FUNCTION "RS485_2" : VOID	// FC 2
VERSION : 0.1
BEGIN
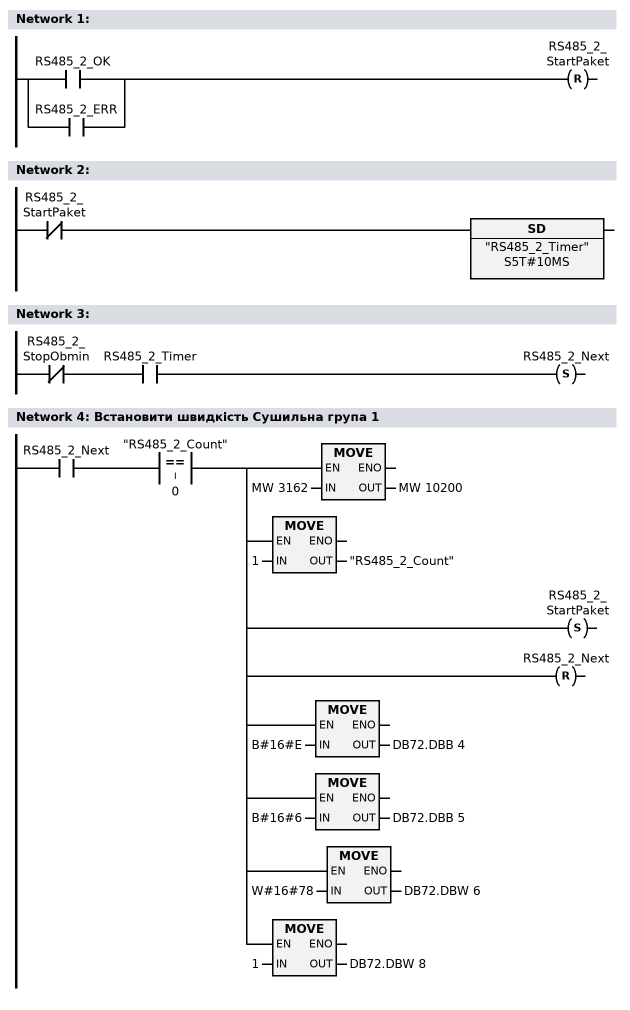
NETWORK
TITLE =
      O     "RS485_2_OK";
      O     "RS485_2_ERR";
      R     "RS485_2_StartPaket";
NETWORK
TITLE =
      AN    "RS485_2_StartPaket";
      L     S5T#10MS;
      SD    "RS485_2_Timer";
NETWORK
TITLE =
      AN    "RS485_2_StopObmin";
      A     "RS485_2_Timer";
      S     "RS485_2_Next";
NETWORK
TITLE = Встановити швидкість Сушильна група 1
      A     "RS485_2_Next";
      A(;
      L     "RS485_2_Count";
      L     0;
      ==I;
      );
      =     L 0.0;
      A     L 0.0;
      JNB   _001;
      L     MW 3162;
      T     MW 10200;
_001: NOP   0;
      A     L 0.0;
      JNB   _002;
      L     1;
      T     "RS485_2_Count";
_002: NOP   0;
      A     L 0.0;
      BLD   102;
      S     "RS485_2_StartPaket";
      A     L 0.0;
      BLD   102;
      R     "RS485_2_Next";
      A     L 0.0;
      JNB   _003;
      L     B#16#E;
      T     DB72.DBB 4;
_003: NOP   0;
      A     L 0.0;
      JNB   _004;
      L     B#16#6;
      T     DB72.DBB 5;
_004: NOP   0;
      A     L 0.0;
      JNB   _005;
      L     W#16#78;
      T     DB72.DBW 6;
_005: NOP   0;
      A     L 0.0;
      JNB   _006;
      L     1;
      T     DB72.DBW 8;
_006: NOP   0;
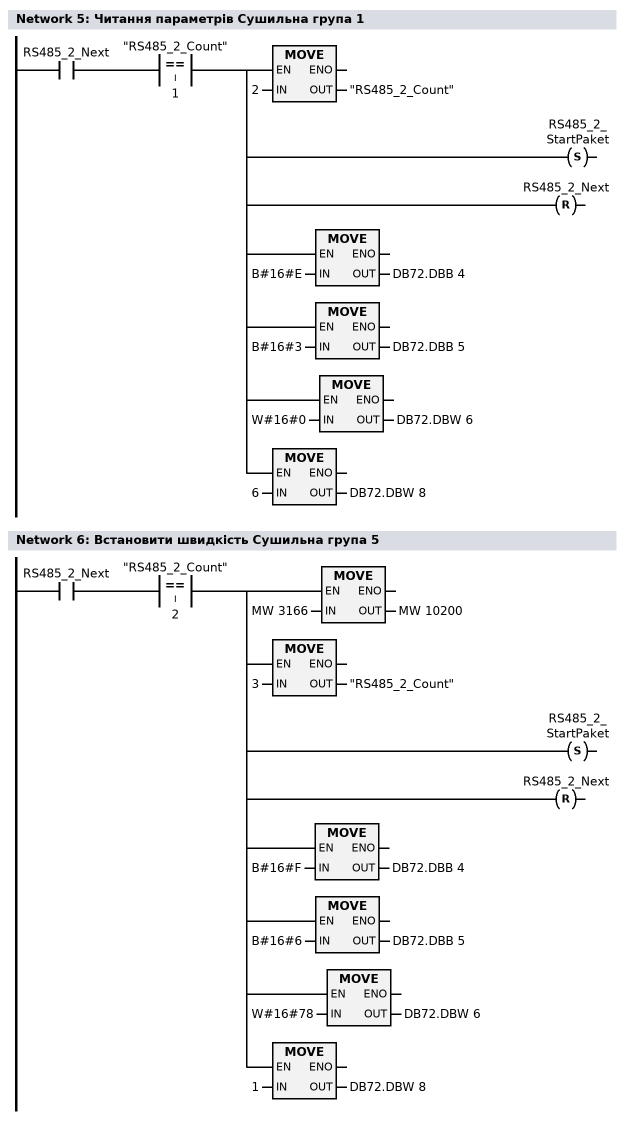
NETWORK
TITLE = Читання параметрів Сушильна група 1
      A     "RS485_2_Next";
      A(;
      L     "RS485_2_Count";
      L     1;
      ==I;
      );
      =     L 0.0;
      A     L 0.0;
      JNB   _007;
      L     2;
      T     "RS485_2_Count";
_007: NOP   0;
      A     L 0.0;
      BLD   102;
      S     "RS485_2_StartPaket";
      A     L 0.0;
      BLD   102;
      R     "RS485_2_Next";
      A     L 0.0;
      JNB   _008;
      L     B#16#E;
      T     DB72.DBB 4;
_008: NOP   0;
      A     L 0.0;
      JNB   _009;
      L     B#16#3;
      T     DB72.DBB 5;
_009: NOP   0;
      A     L 0.0;
      JNB   _00a;
      L     W#16#0;
      T     DB72.DBW 6;
_00a: NOP   0;
      A     L 0.0;
      JNB   _00b;
      L     6;
      T     DB72.DBW 8;
_00b: NOP   0;
NETWORK
TITLE = Встановити швидкість Сушильна група 5
      A     "RS485_2_Next";
      A(;
      L     "RS485_2_Count";
      L     2;
      ==I;
      );
      =     L 0.0;
      A     L 0.0;
      JNB   _00c;
      L     MW 3166;
      T     MW 10200;
_00c: NOP   0;
      A     L 0.0;
      JNB   _00d;
      L     3;
      T     "RS485_2_Count";
_00d: NOP   0;
      A     L 0.0;
      BLD   102;
      S     "RS485_2_StartPaket";
      A     L 0.0;
      BLD   102;
      R     "RS485_2_Next";
      A     L 0.0;
      JNB   _00e;
      L     B#16#F;
      T     DB72.DBB 4;
_00e: NOP   0;
      A     L 0.0;
      JNB   _00f;
      L     B#16#6;
      T     DB72.DBB 5;
_00f: NOP   0;
      A     L 0.0;
      JNB   _010;
      L     W#16#78;
      T     DB72.DBW 6;
_010: NOP   0;
      A     L 0.0;
      JNB   _011;
      L     1;
      T     DB72.DBW 8;
_011: NOP   0;
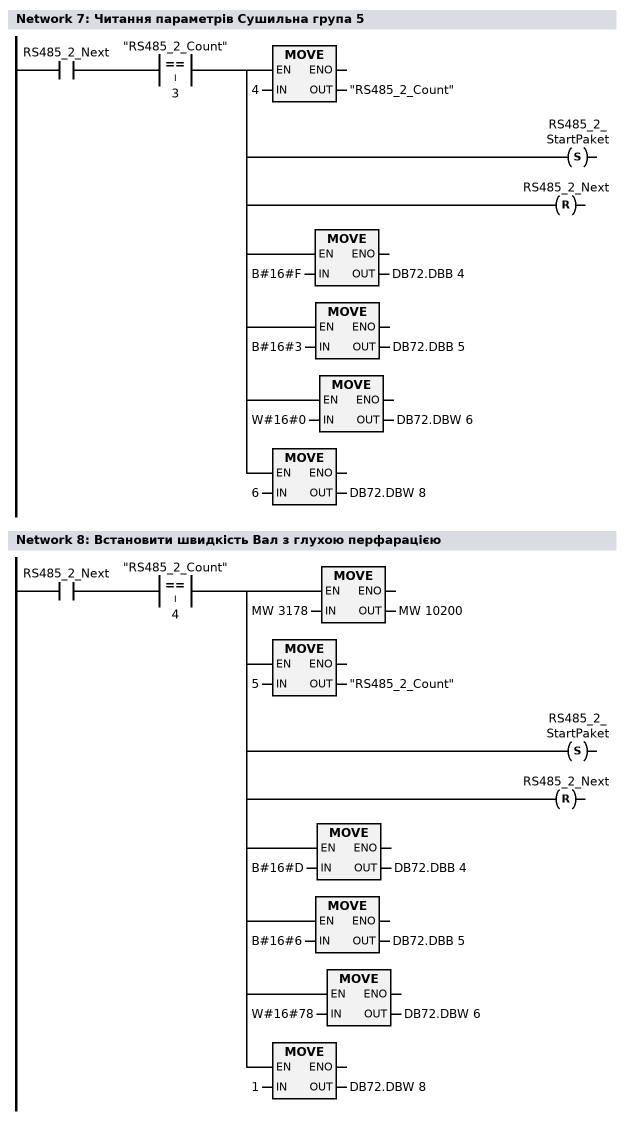
NETWORK
TITLE = Читання параметрів Сушильна група 5
      A     "RS485_2_Next";
      A(;
      L     "RS485_2_Count";
      L     3;
      ==I;
      );
      =     L 0.0;
      A     L 0.0;
      JNB   _012;
      L     4;
      T     "RS485_2_Count";
_012: NOP   0;
      A     L 0.0;
      BLD   102;
      S     "RS485_2_StartPaket";
      A     L 0.0;
      BLD   102;
      R     "RS485_2_Next";
      A     L 0.0;
      JNB   _013;
      L     B#16#F;
      T     DB72.DBB 4;
_013: NOP   0;
      A     L 0.0;
      JNB   _014;
      L     B#16#3;
      T     DB72.DBB 5;
_014: NOP   0;
      A     L 0.0;
      JNB   _015;
      L     W#16#0;
      T     DB72.DBW 6;
_015: NOP   0;
      A     L 0.0;
      JNB   _016;
      L     6;
      T     DB72.DBW 8;
_016: NOP   0;
NETWORK
TITLE = Встановити швидкість Вал з глухою перфарацією
      A     "RS485_2_Next";
      A(;
      L     "RS485_2_Count";
      L     4;
      ==I;
      );
      =     L 0.0;
      A     L 0.0;
      JNB   _017;
      L     MW 3178;
      T     MW 10200;
_017: NOP   0;
      A     L 0.0;
      JNB   _018;
      L     5;
      T     "RS485_2_Count";
_018: NOP   0;
      A     L 0.0;
      BLD   102;
      S     "RS485_2_StartPaket";
      A     L 0.0;
      BLD   102;
      R     "RS485_2_Next";
      A     L 0.0;
      JNB   _019;
      L     B#16#D;
      T     DB72.DBB 4;
_019: NOP   0;
      A     L 0.0;
      JNB   _01a;
      L     B#16#6;
      T     DB72.DBB 5;
_01a: NOP   0;
      A     L 0.0;
      JNB   _01b;
      L     W#16#78;
      T     DB72.DBW 6;
_01b: NOP   0;
      A     L 0.0;
      JNB   _01c;
      L     1;
      T     DB72.DBW 8;
_01c: NOP   0;
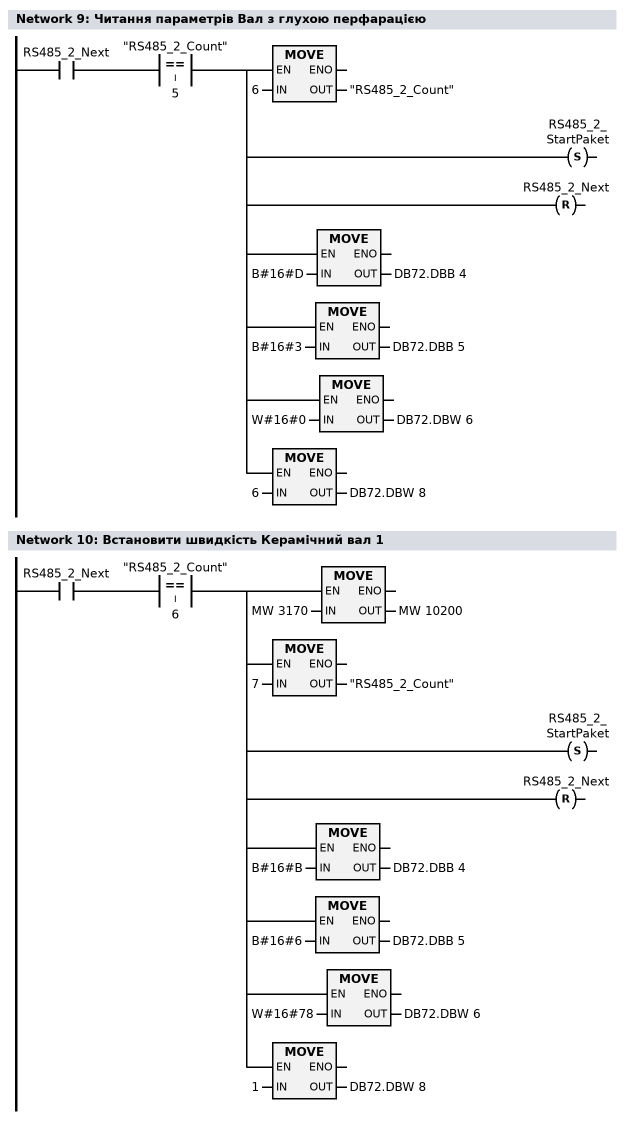
NETWORK
TITLE = Читання параметрів Вал з глухою перфарацією
      A     "RS485_2_Next";
      A(;
      L     "RS485_2_Count";
      L     5;
      ==I;
      );
      =     L 0.0;
      A     L 0.0;
      JNB   _01d;
      L     6;
      T     "RS485_2_Count";
_01d: NOP   0;
      A     L 0.0;
      BLD   102;
      S     "RS485_2_StartPaket";
      A     L 0.0;
      BLD   102;
      R     "RS485_2_Next";
      A     L 0.0;
      JNB   _01e;
      L     B#16#D;
      T     DB72.DBB 4;
_01e: NOP   0;
      A     L 0.0;
      JNB   _01f;
      L     B#16#3;
      T     DB72.DBB 5;
_01f: NOP   0;
      A     L 0.0;
      JNB   _020;
      L     W#16#0;
      T     DB72.DBW 6;
_020: NOP   0;
      A     L 0.0;
      JNB   _021;
      L     6;
      T     DB72.DBW 8;
_021: NOP   0;
NETWORK
TITLE = Встановити швидкість Керамічний вал 1
      A     "RS485_2_Next";
      A(;
      L     "RS485_2_Count";
      L     6;
      ==I;
      );
      =     L 0.0;
      A     L 0.0;
      JNB   _022;
      L     MW 3170;
      T     MW 10200;
_022: NOP   0;
      A     L 0.0;
      JNB   _023;
      L     7;
      T     "RS485_2_Count";
_023: NOP   0;
      A     L 0.0;
      BLD   102;
      S     "RS485_2_StartPaket";
      A     L 0.0;
      BLD   102;
      R     "RS485_2_Next";
      A     L 0.0;
      JNB   _024;
      L     B#16#B;
      T     DB72.DBB 4;
_024: NOP   0;
      A     L 0.0;
      JNB   _025;
      L     B#16#6;
      T     DB72.DBB 5;
_025: NOP   0;
      A     L 0.0;
      JNB   _026;
      L     W#16#78;
      T     DB72.DBW 6;
_026: NOP   0;
      A     L 0.0;
      JNB   _027;
      L     1;
      T     DB72.DBW 8;
_027: NOP   0;
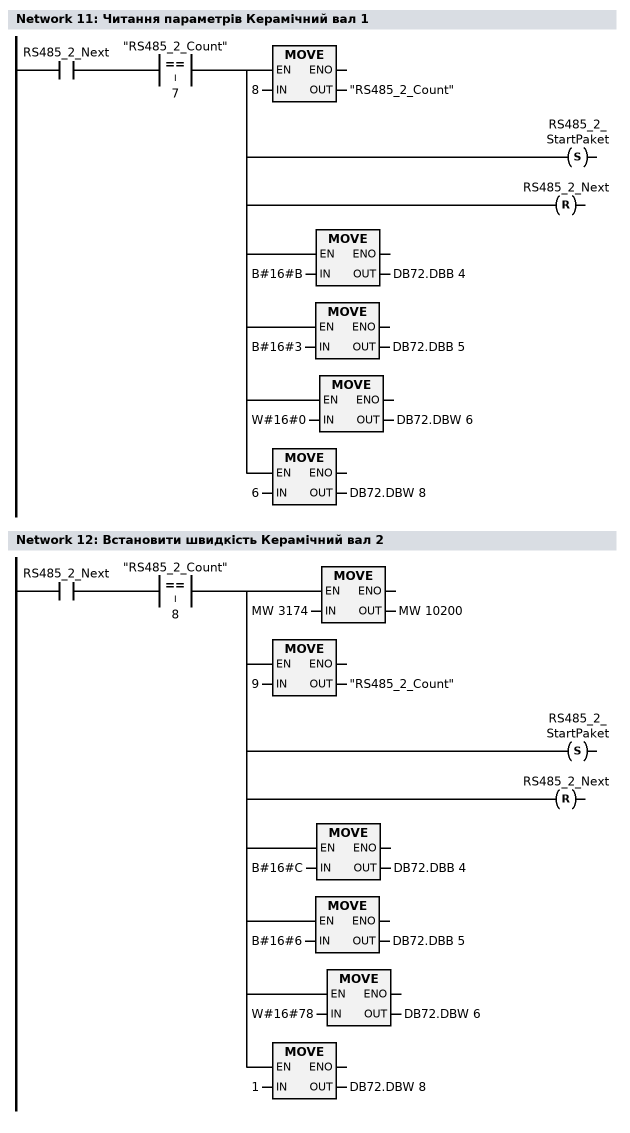
NETWORK
TITLE = Читання параметрів Керамічний вал 1
      A     "RS485_2_Next";
      A(;
      L     "RS485_2_Count";
      L     7;
      ==I;
      );
      =     L 0.0;
      A     L 0.0;
      JNB   _028;
      L     8;
      T     "RS485_2_Count";
_028: NOP   0;
      A     L 0.0;
      BLD   102;
      S     "RS485_2_StartPaket";
      A     L 0.0;
      BLD   102;
      R     "RS485_2_Next";
      A     L 0.0;
      JNB   _029;
      L     B#16#B;
      T     DB72.DBB 4;
_029: NOP   0;
      A     L 0.0;
      JNB   _02a;
      L     B#16#3;
      T     DB72.DBB 5;
_02a: NOP   0;
      A     L 0.0;
      JNB   _02b;
      L     W#16#0;
      T     DB72.DBW 6;
_02b: NOP   0;
      A     L 0.0;
      JNB   _02c;
      L     6;
      T     DB72.DBW 8;
_02c: NOP   0;
NETWORK
TITLE = Встановити швидкість Керамічний вал 2
      A     "RS485_2_Next";
      A(;
      L     "RS485_2_Count";
      L     8;
      ==I;
      );
      =     L 0.0;
      A     L 0.0;
      JNB   _046;
      L     MW 3174;
      T     MW 10200;
_046: NOP   0;
      A     L 0.0;
      JNB   _047;
      L     9;
      T     "RS485_2_Count";
_047: NOP   0;
      A     L 0.0;
      BLD   102;
      S     "RS485_2_StartPaket";
      A     L 0.0;
      BLD   102;
      R     "RS485_2_Next";
      A     L 0.0;
      JNB   _048;
      L     B#16#C;
      T     DB72.DBB 4;
_048: NOP   0;
      A     L 0.0;
      JNB   _049;
      L     B#16#6;
      T     DB72.DBB 5;
_049: NOP   0;
      A     L 0.0;
      JNB   _04a;
      L     W#16#78;
      T     DB72.DBW 6;
_04a: NOP   0;
      A     L 0.0;
      JNB   _04b;
      L     1;
      T     DB72.DBW 8;
_04b: NOP   0;
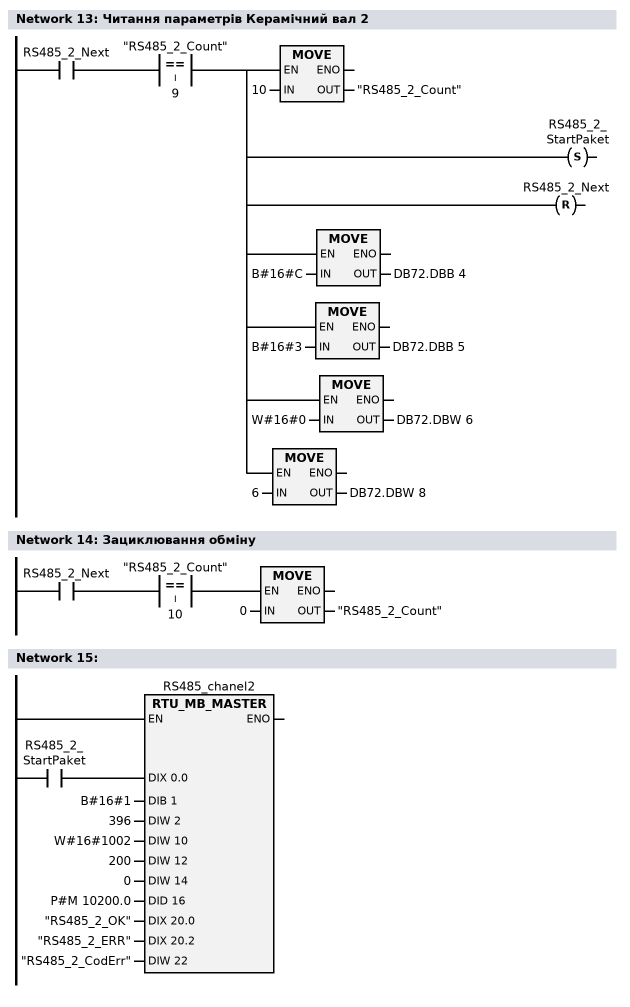
NETWORK
TITLE = Читання параметрів Керамічний вал 2
      A     "RS485_2_Next";
      A(;
      L     "RS485_2_Count";
      L     9;
      ==I;
      );
      =     L 0.0;
      A     L 0.0;
      JNB   _04c;
      L     10;
      T     "RS485_2_Count";
_04c: NOP   0;
      A     L 0.0;
      BLD   102;
      S     "RS485_2_StartPaket";
      A     L 0.0;
      BLD   102;
      R     "RS485_2_Next";
      A     L 0.0;
      JNB   _04d;
      L     B#16#C;
      T     DB72.DBB 4;
_04d: NOP   0;
      A     L 0.0;
      JNB   _04e;
      L     B#16#3;
      T     DB72.DBB 5;
_04e: NOP   0;
      A     L 0.0;
      JNB   _04f;
      L     W#16#0;
      T     DB72.DBW 6;
_04f: NOP   0;
      A     L 0.0;
      JNB   _050;
      L     6;
      T     DB72.DBW 8;
_050: NOP   0;
NETWORK
TITLE = Зациклювання обміну
      A     "RS485_2_Next";
      A(;
      L     "RS485_2_Count";
      L     10;
      ==I;
      );
      JNB   _051;
      L     0;
      T     "RS485_2_Count";
_051: NOP   0;
NETWORK
TITLE =
      A     "RS485_2_StartPaket";
      =     L 0.0;
      BLD   103;
      CALL  "RTU_MB_MASTER" , "RS485_chanel2" (
           DIX 0.0                  := L 0.0,
           DIB 1                    := B#16#1,
           DIW 2                    := 396,
           DIW 10                   := W#16#1002,
           DIW 12                   := 200,
           DIW 14                   := 0,
           DID 16                   := P#M 10200.0,
           DIX 20.0                 := "RS485_2_OK",
           DIX 20.2                 := "RS485_2_ERR",
           DIW 22                   := "RS485_2_CodErr");
      NOP   0;
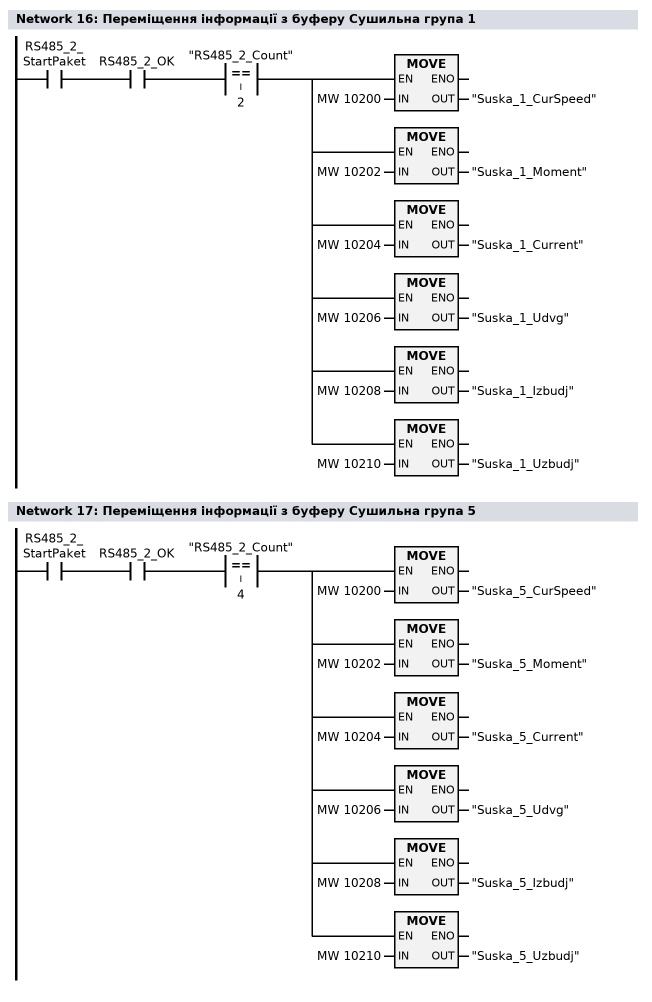
NETWORK
TITLE = Переміщення інформації з буферу Сушильна група 1
      A     "RS485_2_StartPaket";
      A     "RS485_2_OK";
      A(;
      L     "RS485_2_Count";
      L     2;
      ==I;
      );
      =     L 0.0;
      A     L 0.0;
      JNB   _052;
      L     MW 10200;
      T     "Suska_1_CurSpeed";
_052: NOP   0;
      A     L 0.0;
      JNB   _053;
      L     MW 10202;
      T     "Suska_1_Moment";
_053: NOP   0;
      A     L 0.0;
      JNB   _054;
      L     MW 10204;
      T     "Suska_1_Current";
_054: NOP   0;
      A     L 0.0;
      JNB   _055;
      L     MW 10206;
      T     "Suska_1_Udvg";
_055: NOP   0;
      A     L 0.0;
      JNB   _056;
      L     MW 10208;
      T     "Suska_1_Izbudj";
_056: NOP   0;
      A     L 0.0;
      JNB   _057;
      L     MW 10210;
      T     "Suska_1_Uzbudj";
_057: NOP   0;
NETWORK
TITLE = Переміщення інформації з буферу Сушильна група 5
      A     "RS485_2_StartPaket";
      A     "RS485_2_OK";
      A(;
      L     "RS485_2_Count";
      L     4;
      ==I;
      );
      =     L 0.0;
      A     L 0.0;
      JNB   _058;
      L     MW 10200;
      T     "Suska_5_CurSpeed";
_058: NOP   0;
      A     L 0.0;
      JNB   _059;
      L     MW 10202;
      T     "Suska_5_Moment";
_059: NOP   0;
      A     L 0.0;
      JNB   _05a;
      L     MW 10204;
      T     "Suska_5_Current";
_05a: NOP   0;
      A     L 0.0;
      JNB   _05b;
      L     MW 10206;
      T     "Suska_5_Udvg";
_05b: NOP   0;
      A     L 0.0;
      JNB   _05c;
      L     MW 10208;
      T     "Suska_5_Izbudj";
_05c: NOP   0;
      A     L 0.0;
      JNB   _05d;
      L     MW 10210;
      T     "Suska_5_Uzbudj";
_05d: NOP   0;
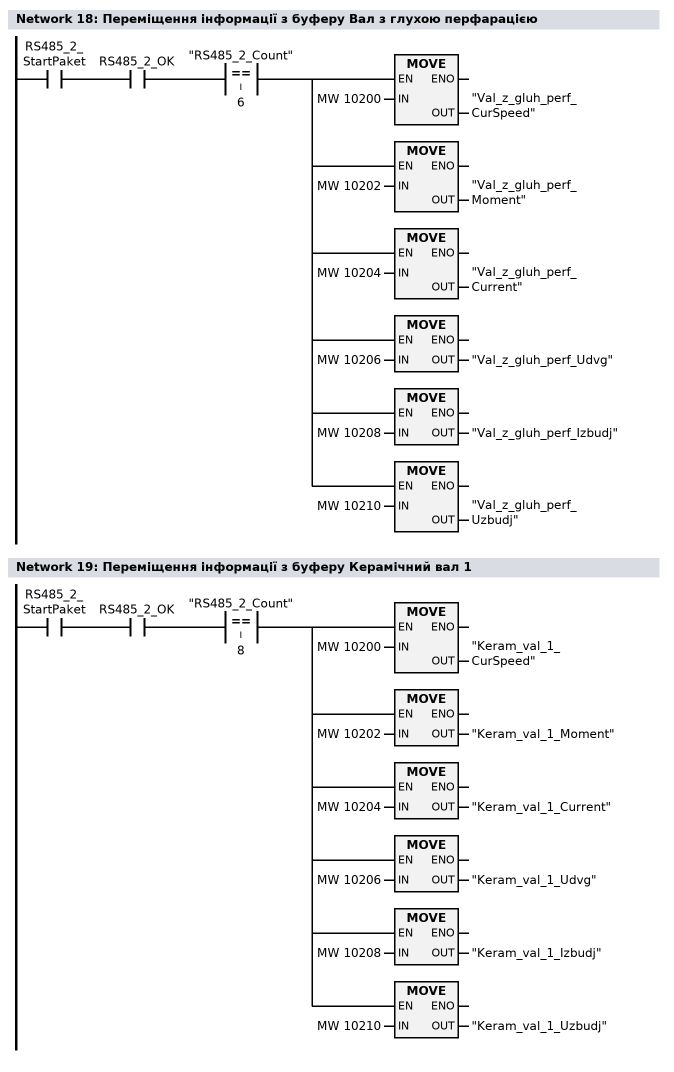
NETWORK
TITLE = Переміщення інформації з буферу Вал з глухою перфарацією
      A     "RS485_2_StartPaket";
      A     "RS485_2_OK";
      A(;
      L     "RS485_2_Count";
      L     6;
      ==I;
      );
      =     L 0.0;
      A     L 0.0;
      JNB   _05e;
      L     MW 10200;
      T     "Val_z_gluh_perf_CurSpeed";
_05e: NOP   0;
      A     L 0.0;
      JNB   _05f;
      L     MW 10202;
      T     "Val_z_gluh_perf_Moment";
_05f: NOP   0;
      A     L 0.0;
      JNB   _060;
      L     MW 10204;
      T     "Val_z_gluh_perf_Current";
_060: NOP   0;
      A     L 0.0;
      JNB   _061;
      L     MW 10206;
      T     "Val_z_gluh_perf_Udvg";
_061: NOP   0;
      A     L 0.0;
      JNB   _062;
      L     MW 10208;
      T     "Val_z_gluh_perf_Izbudj";
_062: NOP   0;
      A     L 0.0;
      JNB   _063;
      L     MW 10210;
      T     "Val_z_gluh_perf_Uzbudj";
_063: NOP   0;
NETWORK
TITLE = Переміщення інформації з буферу Керамічний вал 1
      A     "RS485_2_StartPaket";
      A     "RS485_2_OK";
      A(;
      L     "RS485_2_Count";
      L     8;
      ==I;
      );
      =     L 0.0;
      A     L 0.0;
      JNB   _064;
      L     MW 10200;
      T     "Keram_val_1_CurSpeed";
_064: NOP   0;
      A     L 0.0;
      JNB   _065;
      L     MW 10202;
      T     "Keram_val_1_Moment";
_065: NOP   0;
      A     L 0.0;
      JNB   _066;
      L     MW 10204;
      T     "Keram_val_1_Current";
_066: NOP   0;
      A     L 0.0;
      JNB   _067;
      L     MW 10206;
      T     "Keram_val_1_Udvg";
_067: NOP   0;
      A     L 0.0;
      JNB   _068;
      L     MW 10208;
      T     "Keram_val_1_Izbudj";
_068: NOP   0;
      A     L 0.0;
      JNB   _069;
      L     MW 10210;
      T     "Keram_val_1_Uzbudj";
_069: NOP   0;
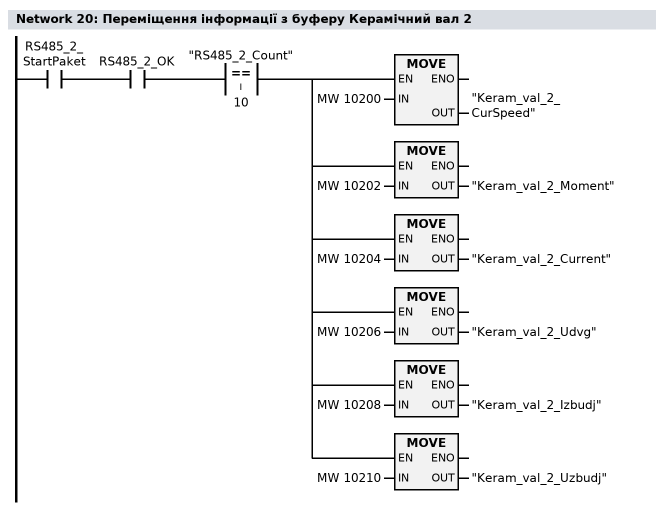
NETWORK
TITLE = Переміщення інформації з буферу Керамічний вал 2
      A     "RS485_2_StartPaket";
      A     "RS485_2_OK";
      A(;
      L     "RS485_2_Count";
      L     10;
      ==I;
      );
      =     L 0.0;
      A     L 0.0;
      JNB   _06a;
      L     MW 10200;
      T     "Keram_val_2_CurSpeed";
_06a: NOP   0;
      A     L 0.0;
      JNB   _06b;
      L     MW 10202;
      T     "Keram_val_2_Moment";
_06b: NOP   0;
      A     L 0.0;
      JNB   _06c;
      L     MW 10204;
      T     "Keram_val_2_Current";
_06c: NOP   0;
      A     L 0.0;
      JNB   _06d;
      L     MW 10206;
      T     "Keram_val_2_Udvg";
_06d: NOP   0;
      A     L 0.0;
      JNB   _06e;
      L     MW 10208;
      T     "Keram_val_2_Izbudj";
_06e: NOP   0;
      A     L 0.0;
      JNB   _06f;
      L     MW 10210;
      T     "Keram_val_2_Uzbudj";
_06f: NOP   0;
END_FUNCTION

FUNCTION "RS485_Runchanel3" : VOID	// FC 3
VERSION : 0.1
BEGIN
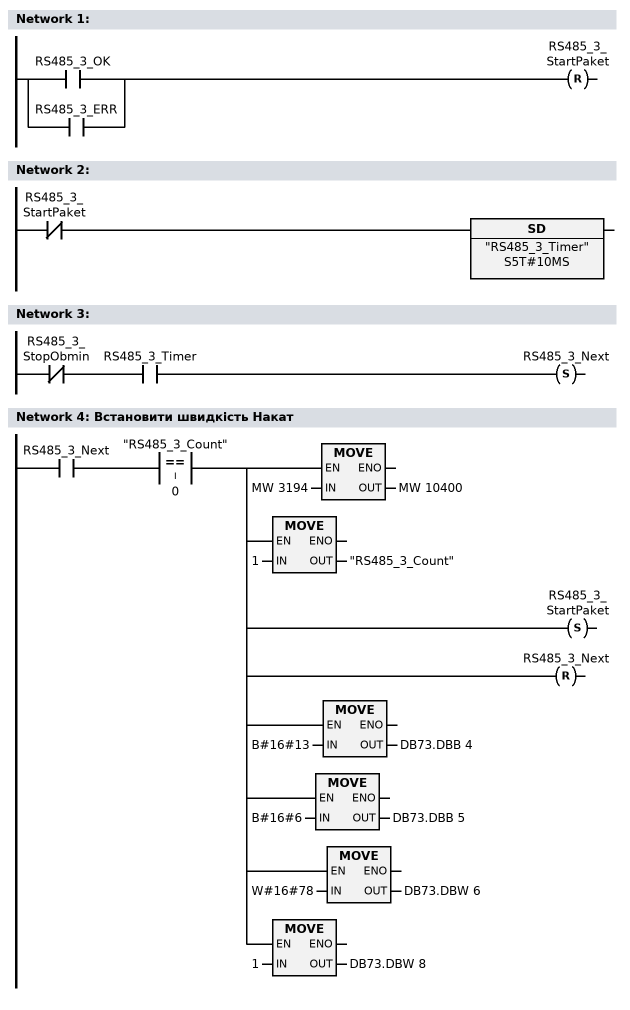
NETWORK
TITLE =
      O     "RS485_3_OK";
      O     "RS485_3_ERR";
      R     "RS485_3_StartPaket";
NETWORK
TITLE =
      AN    "RS485_3_StartPaket";
      L     S5T#10MS;
      SD    "RS485_3_Timer";
NETWORK
TITLE =
      AN    "RS485_3_StopObmin";
      A     "RS485_3_Timer";
      S     "RS485_3_Next";
NETWORK
TITLE = Встановити швидкість Накат
      A     "RS485_3_Next";
      A(;
      L     "RS485_3_Count";
      L     0;
      ==I;
      );
      =     L 0.0;
      A     L 0.0;
      JNB   _001;
      L     MW 3194;
      T     MW 10400;
_001: NOP   0;
      A     L 0.0;
      JNB   _002;
      L     1;
      T     "RS485_3_Count";
_002: NOP   0;
      A     L 0.0;
      BLD   102;
      S     "RS485_3_StartPaket";
      A     L 0.0;
      BLD   102;
      R     "RS485_3_Next";
      A     L 0.0;
      JNB   _003;
      L     B#16#13;
      T     DB73.DBB 4;
_003: NOP   0;
      A     L 0.0;
      JNB   _004;
      L     B#16#6;
      T     DB73.DBB 5;
_004: NOP   0;
      A     L 0.0;
      JNB   _005;
      L     W#16#78;
      T     DB73.DBW 6;
_005: NOP   0;
      A     L 0.0;
      JNB   _006;
      L     1;
      T     DB73.DBW 8;
_006: NOP   0;
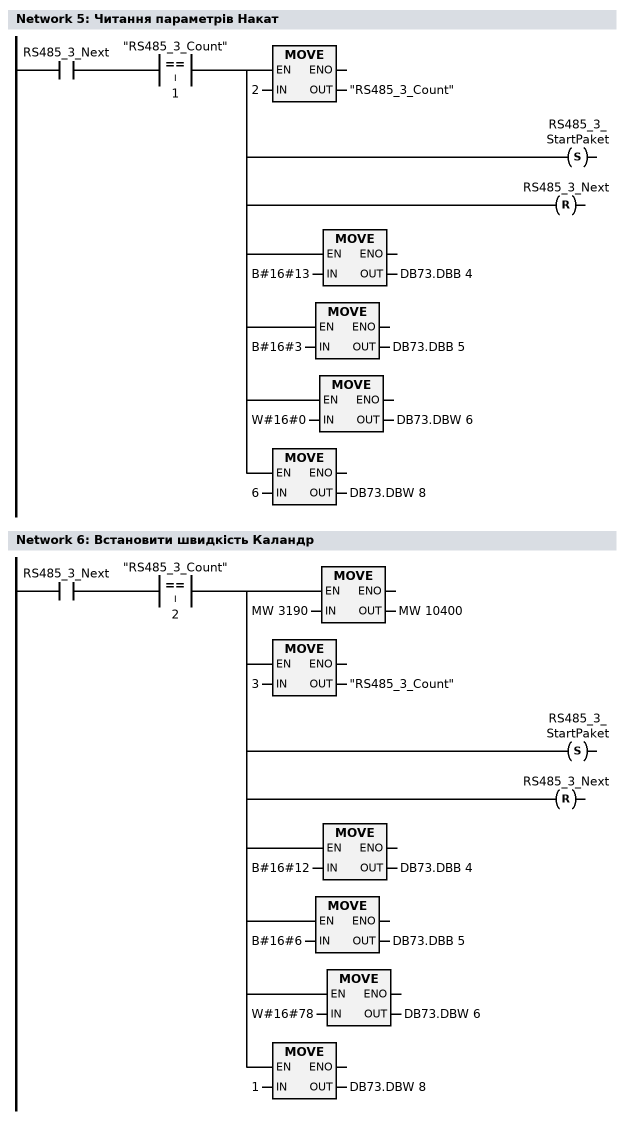
NETWORK
TITLE = Читання параметрів Накат
      A     "RS485_3_Next";
      A(;
      L     "RS485_3_Count";
      L     1;
      ==I;
      );
      =     L 0.0;
      A     L 0.0;
      JNB   _007;
      L     2;
      T     "RS485_3_Count";
_007: NOP   0;
      A     L 0.0;
      BLD   102;
      S     "RS485_3_StartPaket";
      A     L 0.0;
      BLD   102;
      R     "RS485_3_Next";
      A     L 0.0;
      JNB   _008;
      L     B#16#13;
      T     DB73.DBB 4;
_008: NOP   0;
      A     L 0.0;
      JNB   _009;
      L     B#16#3;
      T     DB73.DBB 5;
_009: NOP   0;
      A     L 0.0;
      JNB   _00a;
      L     W#16#0;
      T     DB73.DBW 6;
_00a: NOP   0;
      A     L 0.0;
      JNB   _00b;
      L     6;
      T     DB73.DBW 8;
_00b: NOP   0;
NETWORK
TITLE = Встановити швидкість Каландр
      A     "RS485_3_Next";
      A(;
      L     "RS485_3_Count";
      L     2;
      ==I;
      );
      =     L 0.0;
      A     L 0.0;
      JNB   _00c;
      L     MW 3190;
      T     MW 10400;
_00c: NOP   0;
      A     L 0.0;
      JNB   _00d;
      L     3;
      T     "RS485_3_Count";
_00d: NOP   0;
      A     L 0.0;
      BLD   102;
      S     "RS485_3_StartPaket";
      A     L 0.0;
      BLD   102;
      R     "RS485_3_Next";
      A     L 0.0;
      JNB   _00e;
      L     B#16#12;
      T     DB73.DBB 4;
_00e: NOP   0;
      A     L 0.0;
      JNB   _00f;
      L     B#16#6;
      T     DB73.DBB 5;
_00f: NOP   0;
      A     L 0.0;
      JNB   _010;
      L     W#16#78;
      T     DB73.DBW 6;
_010: NOP   0;
      A     L 0.0;
      JNB   _011;
      L     1;
      T     DB73.DBW 8;
_011: NOP   0;
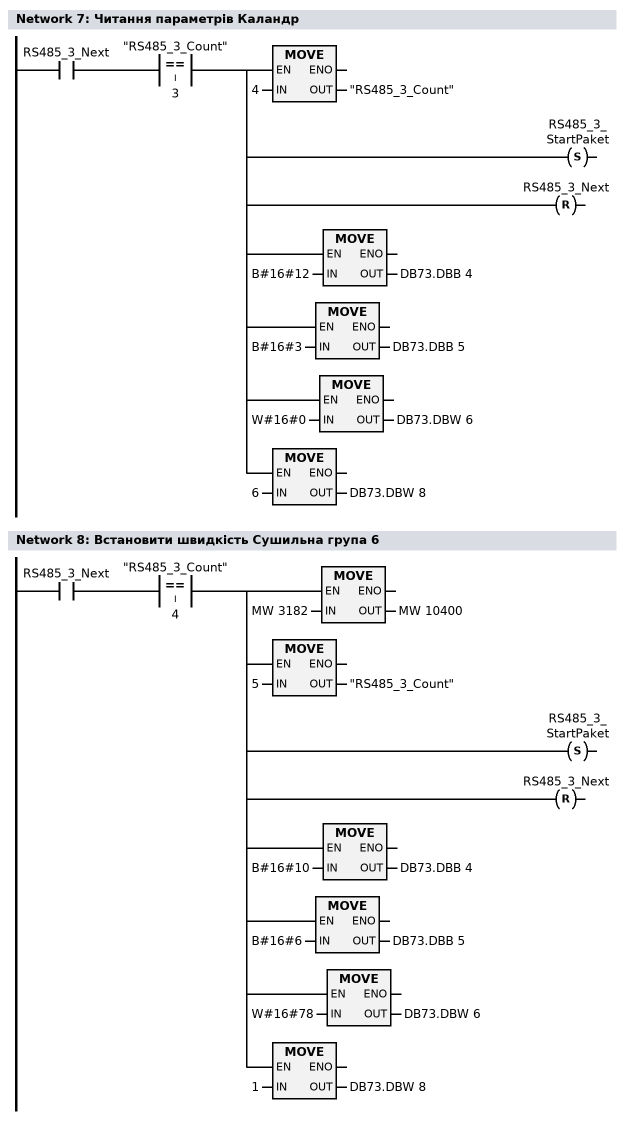
NETWORK
TITLE = Читання параметрів Каландр
      A     "RS485_3_Next";
      A(;
      L     "RS485_3_Count";
      L     3;
      ==I;
      );
      =     L 0.0;
      A     L 0.0;
      JNB   _012;
      L     4;
      T     "RS485_3_Count";
_012: NOP   0;
      A     L 0.0;
      BLD   102;
      S     "RS485_3_StartPaket";
      A     L 0.0;
      BLD   102;
      R     "RS485_3_Next";
      A     L 0.0;
      JNB   _013;
      L     B#16#12;
      T     DB73.DBB 4;
_013: NOP   0;
      A     L 0.0;
      JNB   _014;
      L     B#16#3;
      T     DB73.DBB 5;
_014: NOP   0;
      A     L 0.0;
      JNB   _015;
      L     W#16#0;
      T     DB73.DBW 6;
_015: NOP   0;
      A     L 0.0;
      JNB   _016;
      L     6;
      T     DB73.DBW 8;
_016: NOP   0;
NETWORK
TITLE = Встановити швидкість Сушильна група 6
      A     "RS485_3_Next";
      A(;
      L     "RS485_3_Count";
      L     4;
      ==I;
      );
      =     L 0.0;
      A     L 0.0;
      JNB   _017;
      L     MW 3182;
      T     MW 10400;
_017: NOP   0;
      A     L 0.0;
      JNB   _018;
      L     5;
      T     "RS485_3_Count";
_018: NOP   0;
      A     L 0.0;
      BLD   102;
      S     "RS485_3_StartPaket";
      A     L 0.0;
      BLD   102;
      R     "RS485_3_Next";
      A     L 0.0;
      JNB   _019;
      L     B#16#10;
      T     DB73.DBB 4;
_019: NOP   0;
      A     L 0.0;
      JNB   _01a;
      L     B#16#6;
      T     DB73.DBB 5;
_01a: NOP   0;
      A     L 0.0;
      JNB   _01b;
      L     W#16#78;
      T     DB73.DBW 6;
_01b: NOP   0;
      A     L 0.0;
      JNB   _01c;
      L     1;
      T     DB73.DBW 8;
_01c: NOP   0;
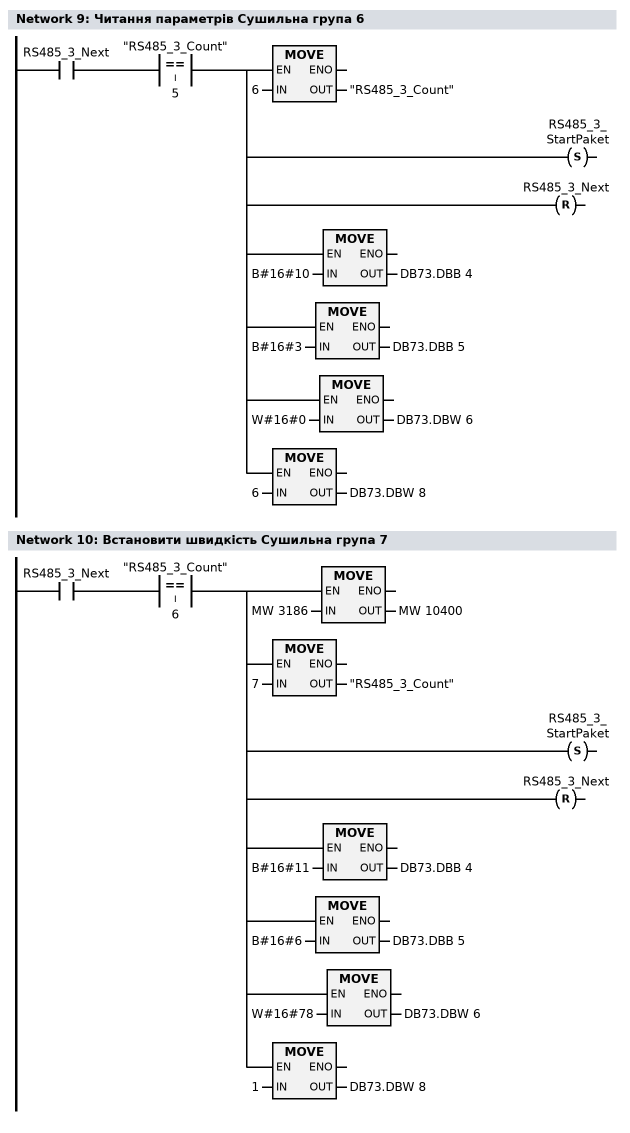
NETWORK
TITLE = Читання параметрів Сушильна група 6
      A     "RS485_3_Next";
      A(;
      L     "RS485_3_Count";
      L     5;
      ==I;
      );
      =     L 0.0;
      A     L 0.0;
      JNB   _01d;
      L     6;
      T     "RS485_3_Count";
_01d: NOP   0;
      A     L 0.0;
      BLD   102;
      S     "RS485_3_StartPaket";
      A     L 0.0;
      BLD   102;
      R     "RS485_3_Next";
      A     L 0.0;
      JNB   _01e;
      L     B#16#10;
      T     DB73.DBB 4;
_01e: NOP   0;
      A     L 0.0;
      JNB   _01f;
      L     B#16#3;
      T     DB73.DBB 5;
_01f: NOP   0;
      A     L 0.0;
      JNB   _020;
      L     W#16#0;
      T     DB73.DBW 6;
_020: NOP   0;
      A     L 0.0;
      JNB   _021;
      L     6;
      T     DB73.DBW 8;
_021: NOP   0;
NETWORK
TITLE = Встановити швидкість Сушильна група 7
      A     "RS485_3_Next";
      A(;
      L     "RS485_3_Count";
      L     6;
      ==I;
      );
      =     L 0.0;
      A     L 0.0;
      JNB   _022;
      L     MW 3186;
      T     MW 10400;
_022: NOP   0;
      A     L 0.0;
      JNB   _023;
      L     7;
      T     "RS485_3_Count";
_023: NOP   0;
      A     L 0.0;
      BLD   102;
      S     "RS485_3_StartPaket";
      A     L 0.0;
      BLD   102;
      R     "RS485_3_Next";
      A     L 0.0;
      JNB   _024;
      L     B#16#11;
      T     DB73.DBB 4;
_024: NOP   0;
      A     L 0.0;
      JNB   _025;
      L     B#16#6;
      T     DB73.DBB 5;
_025: NOP   0;
      A     L 0.0;
      JNB   _026;
      L     W#16#78;
      T     DB73.DBW 6;
_026: NOP   0;
      A     L 0.0;
      JNB   _027;
      L     1;
      T     DB73.DBW 8;
_027: NOP   0;
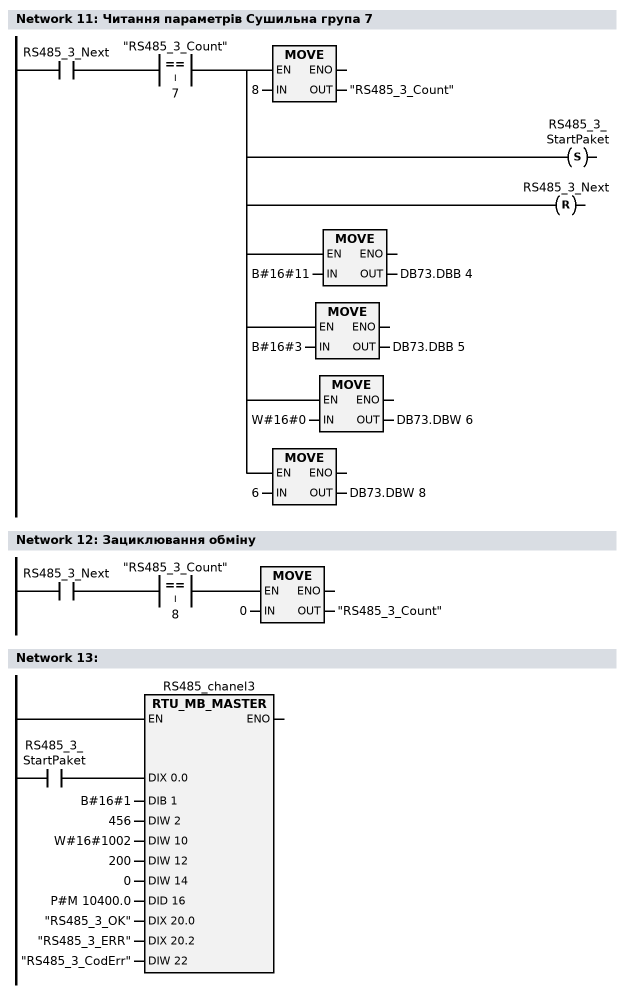
NETWORK
TITLE = Читання параметрів Сушильна група 7
      A     "RS485_3_Next";
      A(;
      L     "RS485_3_Count";
      L     7;
      ==I;
      );
      =     L 0.0;
      A     L 0.0;
      JNB   _028;
      L     8;
      T     "RS485_3_Count";
_028: NOP   0;
      A     L 0.0;
      BLD   102;
      S     "RS485_3_StartPaket";
      A     L 0.0;
      BLD   102;
      R     "RS485_3_Next";
      A     L 0.0;
      JNB   _029;
      L     B#16#11;
      T     DB73.DBB 4;
_029: NOP   0;
      A     L 0.0;
      JNB   _02a;
      L     B#16#3;
      T     DB73.DBB 5;
_02a: NOP   0;
      A     L 0.0;
      JNB   _02b;
      L     W#16#0;
      T     DB73.DBW 6;
_02b: NOP   0;
      A     L 0.0;
      JNB   _02c;
      L     6;
      T     DB73.DBW 8;
_02c: NOP   0;
NETWORK
TITLE = Зациклювання обміну
      A     "RS485_3_Next";
      A(;
      L     "RS485_3_Count";
      L     8;
      ==I;
      );
      JNB   _02d;
      L     0;
      T     "RS485_3_Count";
_02d: NOP   0;
NETWORK
TITLE =
      A     "RS485_3_StartPaket";
      =     L 0.0;
      BLD   103;
      CALL  "RTU_MB_MASTER" , "RS485_chanel3" (
           DIX 0.0                  := L 0.0,
           DIB 1                    := B#16#1,
           DIW 2                    := 456,
           DIW 10                   := W#16#1002,
           DIW 12                   := 200,
           DIW 14                   := 0,
           DID 16                   := P#M 10400.0,
           DIX 20.0                 := "RS485_3_OK",
           DIX 20.2                 := "RS485_3_ERR",
           DIW 22                   := "RS485_3_CodErr");
      NOP   0;
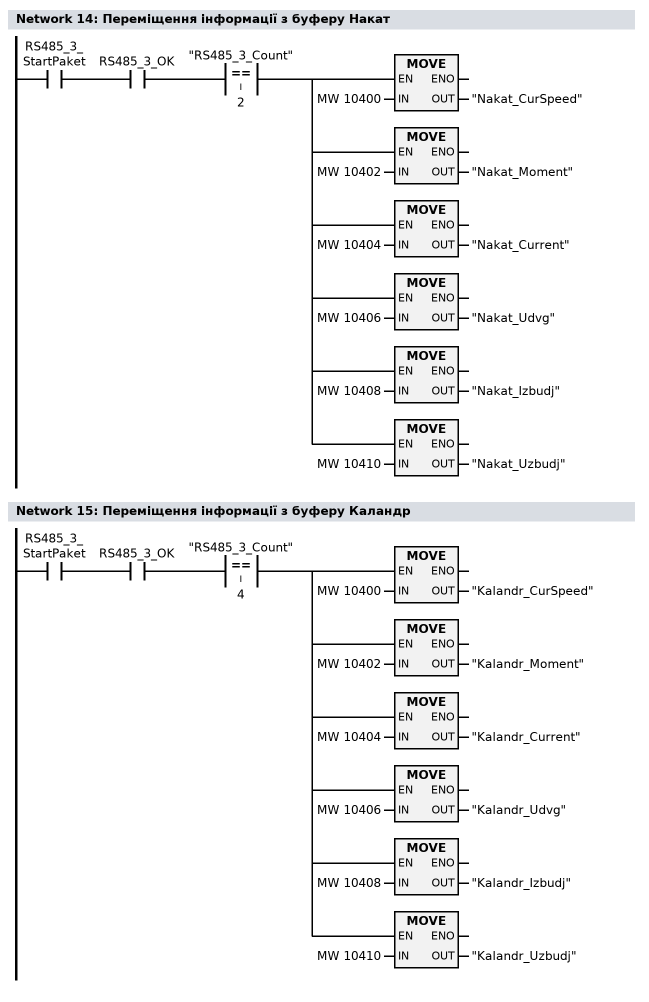
NETWORK
TITLE = Переміщення інформації з буферу Накат
      A     "RS485_3_StartPaket";
      A     "RS485_3_OK";
      A(;
      L     "RS485_3_Count";
      L     2;
      ==I;
      );
      =     L 0.0;
      A     L 0.0;
      JNB   _02e;
      L     MW 10400;
      T     "Nakat_CurSpeed";
_02e: NOP   0;
      A     L 0.0;
      JNB   _02f;
      L     MW 10402;
      T     "Nakat_Moment";
_02f: NOP   0;
      A     L 0.0;
      JNB   _030;
      L     MW 10404;
      T     "Nakat_Current";
_030: NOP   0;
      A     L 0.0;
      JNB   _031;
      L     MW 10406;
      T     "Nakat_Udvg";
_031: NOP   0;
      A     L 0.0;
      JNB   _032;
      L     MW 10408;
      T     "Nakat_Izbudj";
_032: NOP   0;
      A     L 0.0;
      JNB   _033;
      L     MW 10410;
      T     "Nakat_Uzbudj";
_033: NOP   0;
NETWORK
TITLE = Переміщення інформації з буферу Каландр
      A     "RS485_3_StartPaket";
      A     "RS485_3_OK";
      A(;
      L     "RS485_3_Count";
      L     4;
      ==I;
      );
      =     L 0.0;
      A     L 0.0;
      JNB   _034;
      L     MW 10400;
      T     "Kalandr_CurSpeed";
_034: NOP   0;
      A     L 0.0;
      JNB   _035;
      L     MW 10402;
      T     "Kalandr_Moment";
_035: NOP   0;
      A     L 0.0;
      JNB   _036;
      L     MW 10404;
      T     "Kalandr_Current";
_036: NOP   0;
      A     L 0.0;
      JNB   _037;
      L     MW 10406;
      T     "Kalandr_Udvg";
_037: NOP   0;
      A     L 0.0;
      JNB   _038;
      L     MW 10408;
      T     "Kalandr_Izbudj";
_038: NOP   0;
      A     L 0.0;
      JNB   _039;
      L     MW 10410;
      T     "Kalandr_Uzbudj";
_039: NOP   0;
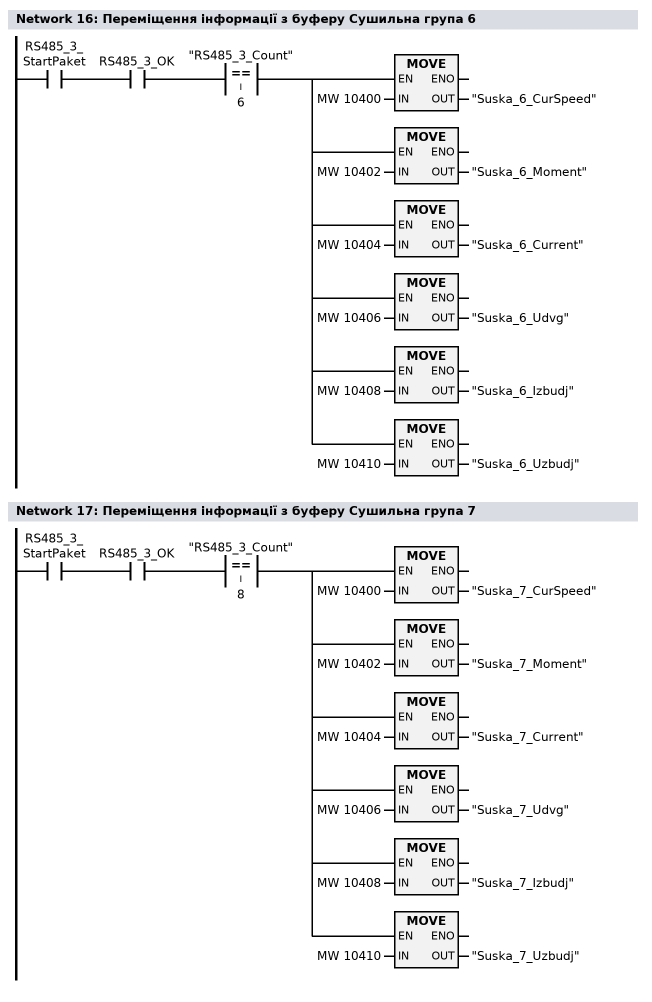
NETWORK
TITLE = Переміщення інформації з буферу Сушильна група 6
      A     "RS485_3_StartPaket";
      A     "RS485_3_OK";
      A(;
      L     "RS485_3_Count";
      L     6;
      ==I;
      );
      =     L 0.0;
      A     L 0.0;
      JNB   _03a;
      L     MW 10400;
      T     "Suska_6_CurSpeed";
_03a: NOP   0;
      A     L 0.0;
      JNB   _03b;
      L     MW 10402;
      T     "Suska_6_Moment";
_03b: NOP   0;
      A     L 0.0;
      JNB   _03c;
      L     MW 10404;
      T     "Suska_6_Current";
_03c: NOP   0;
      A     L 0.0;
      JNB   _03d;
      L     MW 10406;
      T     "Suska_6_Udvg";
_03d: NOP   0;
      A     L 0.0;
      JNB   _03e;
      L     MW 10408;
      T     "Suska_6_Izbudj";
_03e: NOP   0;
      A     L 0.0;
      JNB   _03f;
      L     MW 10410;
      T     "Suska_6_Uzbudj";
_03f: NOP   0;
NETWORK
TITLE = Переміщення інформації з буферу Сушильна група 7
      A     "RS485_3_StartPaket";
      A     "RS485_3_OK";
      A(;
      L     "RS485_3_Count";
      L     8;
      ==I;
      );
      =     L 0.0;
      A     L 0.0;
      JNB   _040;
      L     MW 10400;
      T     "Suska_7_CurSpeed";
_040: NOP   0;
      A     L 0.0;
      JNB   _041;
      L     MW 10402;
      T     "Suska_7_Moment";
_041: NOP   0;
      A     L 0.0;
      JNB   _042;
      L     MW 10404;
      T     "Suska_7_Current";
_042: NOP   0;
      A     L 0.0;
      JNB   _043;
      L     MW 10406;
      T     "Suska_7_Udvg";
_043: NOP   0;
      A     L 0.0;
      JNB   _044;
      L     MW 10408;
      T     "Suska_7_Izbudj";
_044: NOP   0;
      A     L 0.0;
      JNB   _045;
      L     MW 10410;
      T     "Suska_7_Uzbudj";
_045: NOP   0;
END_FUNCTION

FUNCTION "RS485_RunChanel4" : VOID	// FC 4
//RS485_Unit_4
//
VERSION : 0.1
BEGIN
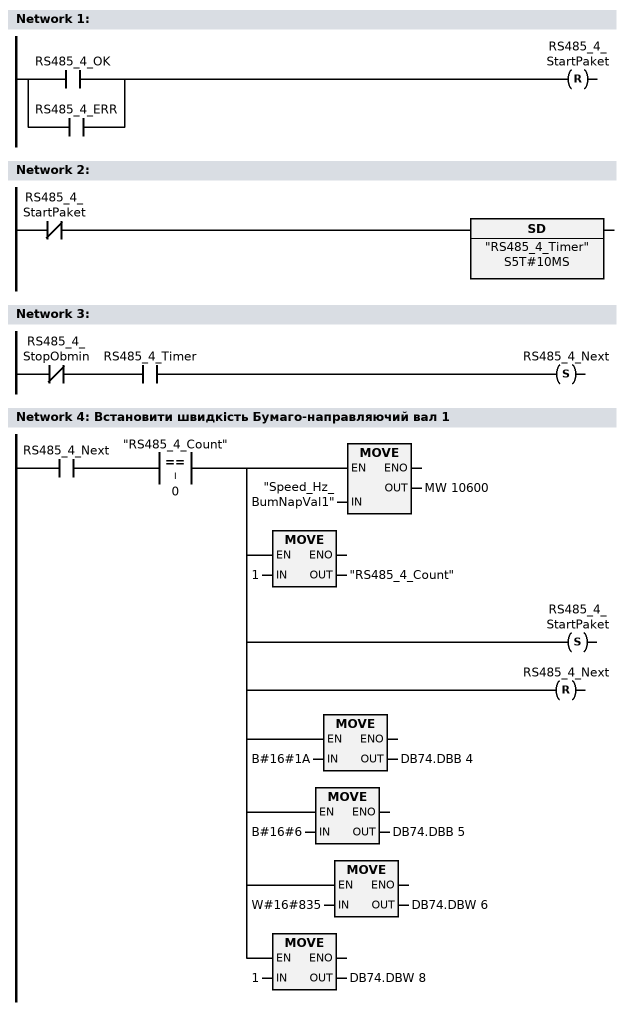
NETWORK
TITLE =
      O     "RS485_4_OK";
      O     "RS485_4_ERR";
      R     "RS485_4_StartPaket";
NETWORK
TITLE =
      AN    "RS485_4_StartPaket";
      L     S5T#10MS;
      SD    "RS485_4_Timer";
NETWORK
TITLE =
      AN    "RS485_4_StopObmin";
      A     "RS485_4_Timer";
      S     "RS485_4_Next";
NETWORK
TITLE = Встановити швидкість Бумаго-направляючий вал 1
      A     "RS485_4_Next";
      A(;
      L     "RS485_4_Count";
      L     0;
      ==I;
      );
      =     L 0.0;
      A     L 0.0;
      JNB   _001;
      L     "Speed_Hz_BumNapVal1";
      T     MW 10600;
_001: NOP   0;
      A     L 0.0;
      JNB   _002;
      L     1;
      T     "RS485_4_Count";
_002: NOP   0;
      A     L 0.0;
      BLD   102;
      S     "RS485_4_StartPaket";
      A     L 0.0;
      BLD   102;
      R     "RS485_4_Next";
      A     L 0.0;
      JNB   _003;
      L     B#16#1A;
      T     DB74.DBB 4;
_003: NOP   0;
      A     L 0.0;
      JNB   _004;
      L     B#16#6;
      T     DB74.DBB 5;
_004: NOP   0;
      A     L 0.0;
      JNB   _005;
      L     W#16#835;
      T     DB74.DBW 6;
_005: NOP   0;
      A     L 0.0;
      JNB   _006;
      L     1;
      T     DB74.DBW 8;
_006: NOP   0;
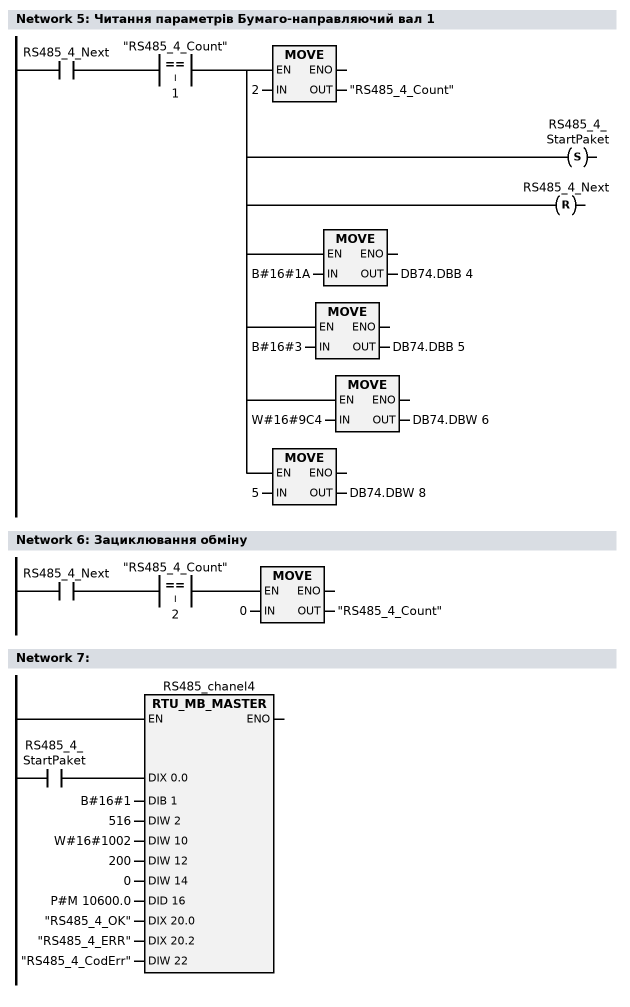
NETWORK
TITLE = Читання параметрів Бумаго-направляючий вал 1
      A     "RS485_4_Next";
      A(;
      L     "RS485_4_Count";
      L     1;
      ==I;
      );
      =     L 0.0;
      A     L 0.0;
      JNB   _007;
      L     2;
      T     "RS485_4_Count";
_007: NOP   0;
      A     L 0.0;
      BLD   102;
      S     "RS485_4_StartPaket";
      A     L 0.0;
      BLD   102;
      R     "RS485_4_Next";
      A     L 0.0;
      JNB   _008;
      L     B#16#1A;
      T     DB74.DBB 4;
_008: NOP   0;
      A     L 0.0;
      JNB   _009;
      L     B#16#3;
      T     DB74.DBB 5;
_009: NOP   0;
      A     L 0.0;
      JNB   _00a;
      L     W#16#9C4;
      T     DB74.DBW 6;
_00a: NOP   0;
      A     L 0.0;
      JNB   _00b;
      L     5;
      T     DB74.DBW 8;
_00b: NOP   0;
NETWORK
TITLE = Зациклювання обміну
      A     "RS485_4_Next";
      A(;
      L     "RS485_4_Count";
      L     2;
      ==I;
      );
      JNB   _00c;
      L     0;
      T     "RS485_4_Count";
_00c: NOP   0;
NETWORK
TITLE =
      A     "RS485_4_StartPaket";
      =     L 0.0;
      BLD   103;
      CALL  "RTU_MB_MASTER" , "RS485_chanel4" (
           DIX 0.0                  := L 0.0,
           DIB 1                    := B#16#1,
           DIW 2                    := 516,
           DIW 10                   := W#16#1002,
           DIW 12                   := 200,
           DIW 14                   := 0,
           DID 16                   := P#M 10600.0,
           DIX 20.0                 := "RS485_4_OK",
           DIX 20.2                 := "RS485_4_ERR",
           DIW 22                   := "RS485_4_CodErr");
      NOP   0;
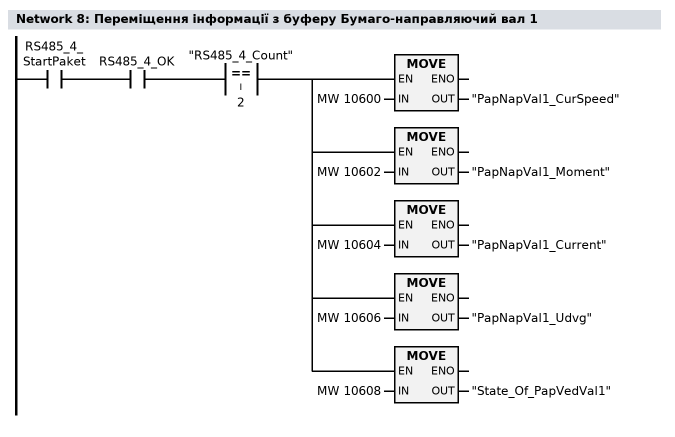
NETWORK
TITLE = Переміщення інформації з буферу Бумаго-направляючий вал 1
      A     "RS485_4_StartPaket";
      A     "RS485_4_OK";
      A(;
      L     "RS485_4_Count";
      L     2;
      ==I;
      );
      =     L 0.0;
      A     L 0.0;
      JNB   _00d;
      L     MW 10600;
      T     "PapNapVal1_CurSpeed";
_00d: NOP   0;
      A     L 0.0;
      JNB   _00e;
      L     MW 10602;
      T     "PapNapVal1_Moment";
_00e: NOP   0;
      A     L 0.0;
      JNB   _00f;
      L     MW 10604;
      T     "PapNapVal1_Current";
_00f: NOP   0;
      A     L 0.0;
      JNB   _010;
      L     MW 10606;
      T     "PapNapVal1_Udvg";
_010: NOP   0;
      A     L 0.0;
      JNB   _011;
      L     MW 10608;
      T     "State_Of_PapVedVal1";
_011: NOP   0;
END_FUNCTION

FUNCTION "Speed_Calculation" : VOID	// FC 10
VERSION : 0.1
VAR_TEMP
  Speed_1R : REAL ;
END_VAR
BEGIN
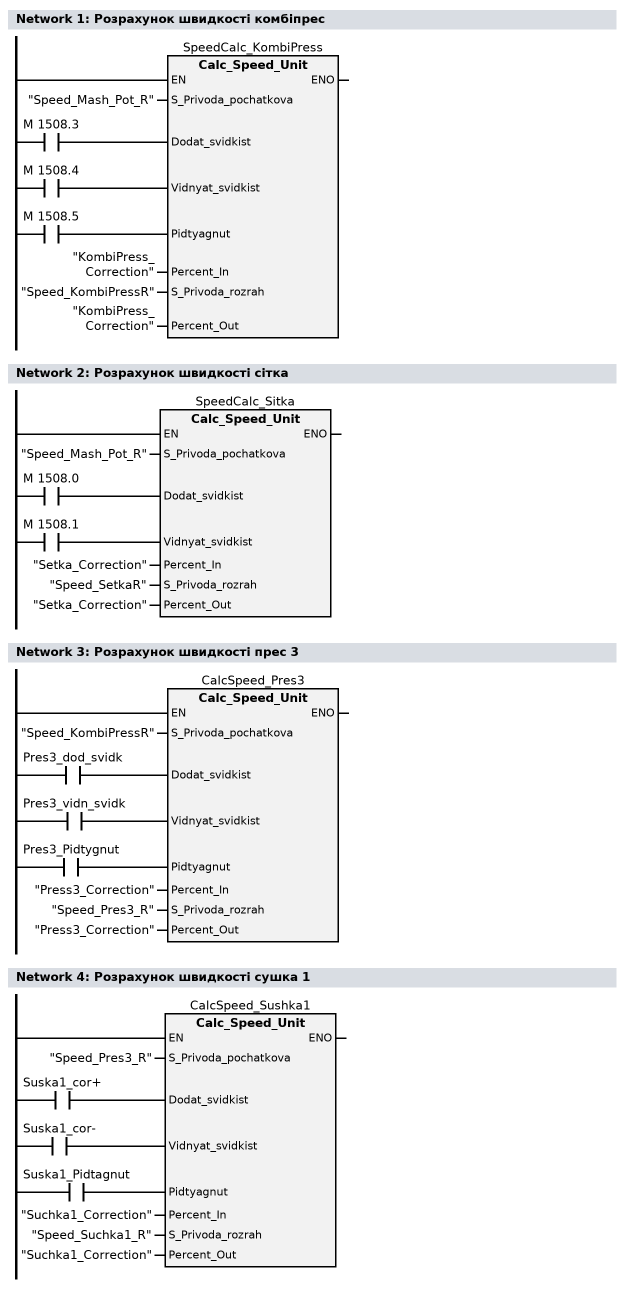
NETWORK
TITLE = Розрахунок швидкості комбіпрес
      A     M 1508.3;
      =     L 4.0;
      BLD   103;
      A     M 1508.4;
      =     L 4.1;
      BLD   103;
      A     M 1508.5;
      =     L 4.2;
      BLD   103;
      CALL  "Calc_Speed_Unit" , "SpeedCalc_KombiPress" (
           S_Privoda_pochatkova     := "Speed_Mash_Pot_R",
           Dodat_svidkist           := L 4.0,
           Vidnyat_svidkist         := L 4.1,
           Pidtyagnut               := L 4.2,
           Percent_In               := "KombiPress_Correction",
           S_Privoda_rozrah         := "Speed_KombiPressR",
           Percent_Out              := "KombiPress_Correction");
      NOP   0;
NETWORK
TITLE = Розрахунок швидкості сітка
      A     M 1508.0;
      =     L 4.0;
      BLD   103;
      A     M 1508.1;
      =     L 4.1;
      BLD   103;
      CALL  "Calc_Speed_Unit" , "SpeedCalc_Sitka" (
           S_Privoda_pochatkova     := "Speed_Mash_Pot_R",
           Dodat_svidkist           := L 4.0,
           Vidnyat_svidkist         := L 4.1,
           Percent_In               := "Setka_Correction",
           S_Privoda_rozrah         := "Speed_SetkaR",
           Percent_Out              := "Setka_Correction");
      NOP   0;
NETWORK
TITLE = Розрахунок швидкості прес 3
      A     "Pres3_dod_svidk";
      =     L 4.0;
      BLD   103;
      A     "Pres3_vidn_svidk";
      =     L 4.1;
      BLD   103;
      A     "Pres3_Pidtygnut";
      =     L 4.2;
      BLD   103;
      CALL  "Calc_Speed_Unit" , "CalcSpeed_Pres3" (
           S_Privoda_pochatkova     := "Speed_KombiPressR",
           Dodat_svidkist           := L 4.0,
           Vidnyat_svidkist         := L 4.1,
           Pidtyagnut               := L 4.2,
           Percent_In               := "Press3_Correction",
           S_Privoda_rozrah         := "Speed_Pres3_R",
           Percent_Out              := "Press3_Correction");
      NOP   0;
NETWORK
TITLE = Розрахунок швидкості сушка 1
      A     "Suska1_cor+";
      =     L 4.0;
      BLD   103;
      A     "Suska1_cor-";
      =     L 4.1;
      BLD   103;
      A     "Suska1_Pidtagnut";
      =     L 4.2;
      BLD   103;
      CALL  "Calc_Speed_Unit" , "CalcSpeed_Sushka1" (
           S_Privoda_pochatkova     := "Speed_Pres3_R",
           Dodat_svidkist           := L 4.0,
           Vidnyat_svidkist         := L 4.1,
           Pidtyagnut               := L 4.2,
           Percent_In               := "Suchka1_Correction",
           S_Privoda_rozrah         := "Speed_Suchka1_R",
           Percent_Out              := "Suchka1_Correction");
      NOP   0;
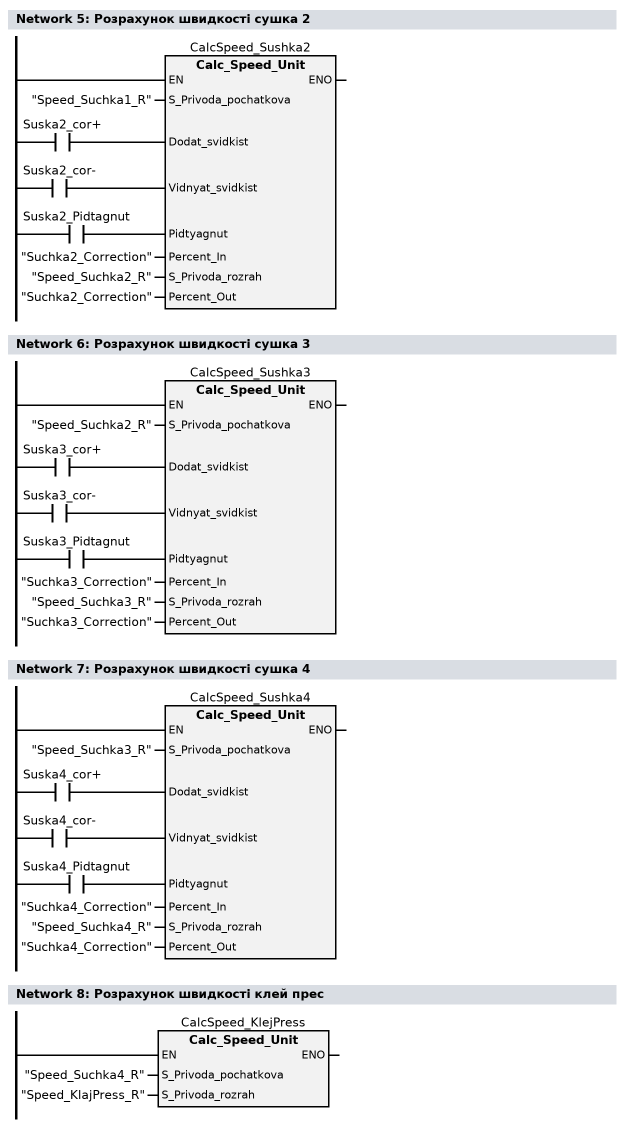
NETWORK
TITLE = Розрахунок швидкості сушка 2
      A     "Suska2_cor+";
      =     L 4.0;
      BLD   103;
      A     "Suska2_cor-";
      =     L 4.1;
      BLD   103;
      A     "Suska2_Pidtagnut";
      =     L 4.2;
      BLD   103;
      CALL  "Calc_Speed_Unit" , "CalcSpeed_Sushka2" (
           S_Privoda_pochatkova     := "Speed_Suchka1_R",
           Dodat_svidkist           := L 4.0,
           Vidnyat_svidkist         := L 4.1,
           Pidtyagnut               := L 4.2,
           Percent_In               := "Suchka2_Correction",
           S_Privoda_rozrah         := "Speed_Suchka2_R",
           Percent_Out              := "Suchka2_Correction");
      NOP   0;
NETWORK
TITLE = Розрахунок швидкості сушка 3
      A     "Suska3_cor+";
      =     L 4.0;
      BLD   103;
      A     "Suska3_cor-";
      =     L 4.1;
      BLD   103;
      A     "Suska3_Pidtagnut";
      =     L 4.2;
      BLD   103;
      CALL  "Calc_Speed_Unit" , "CalcSpeed_Sushka3" (
           S_Privoda_pochatkova     := "Speed_Suchka2_R",
           Dodat_svidkist           := L 4.0,
           Vidnyat_svidkist         := L 4.1,
           Pidtyagnut               := L 4.2,
           Percent_In               := "Suchka3_Correction",
           S_Privoda_rozrah         := "Speed_Suchka3_R",
           Percent_Out              := "Suchka3_Correction");
      NOP   0;
NETWORK
TITLE = Розрахунок швидкості сушка 4
      A     "Suska4_cor+";
      =     L 4.0;
      BLD   103;
      A     "Suska4_cor-";
      =     L 4.1;
      BLD   103;
      A     "Suska4_Pidtagnut";
      =     L 4.2;
      BLD   103;
      CALL  "Calc_Speed_Unit" , "CalcSpeed_Sushka4" (
           S_Privoda_pochatkova     := "Speed_Suchka3_R",
           Dodat_svidkist           := L 4.0,
           Vidnyat_svidkist         := L 4.1,
           Pidtyagnut               := L 4.2,
           Percent_In               := "Suchka4_Correction",
           S_Privoda_rozrah         := "Speed_Suchka4_R",
           Percent_Out              := "Suchka4_Correction");
      NOP   0;
NETWORK
TITLE = Розрахунок швидкості клей прес
      CALL  "Calc_Speed_Unit" , "CalcSpeed_KlejPress" (
           S_Privoda_pochatkova     := "Speed_Suchka4_R",
           S_Privoda_rozrah         := "Speed_KlajPress_R");
      NOP   0;
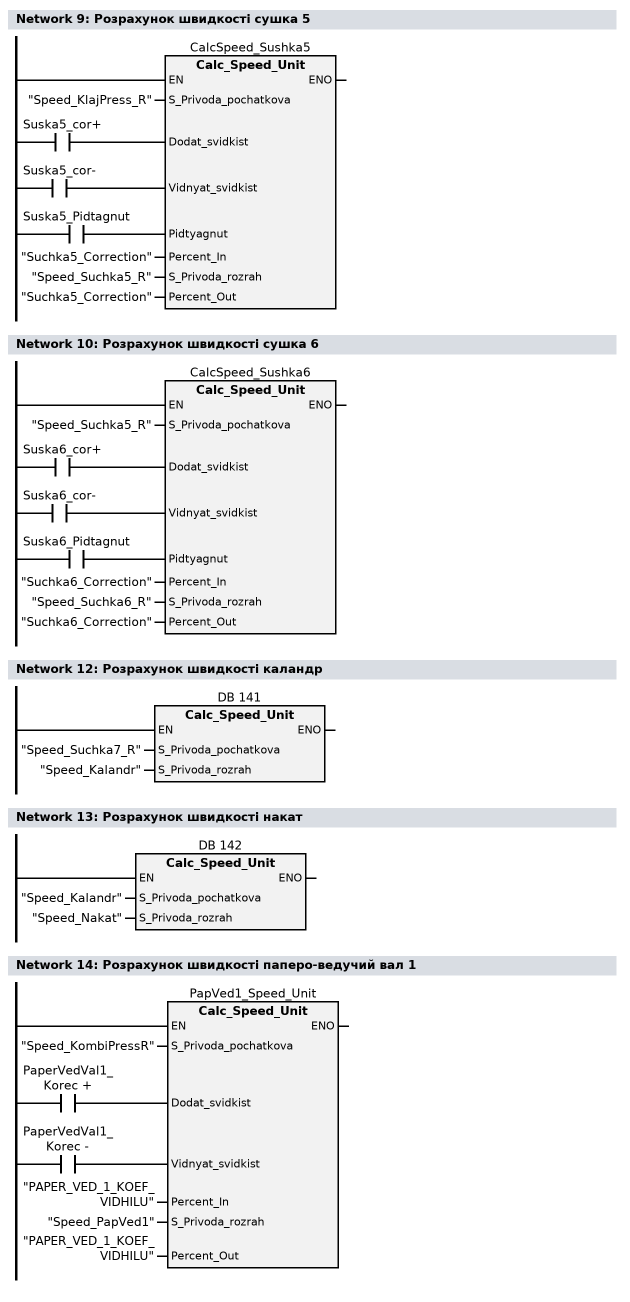
NETWORK
TITLE = Розрахунок швидкості сушка 5
      A     "Suska5_cor+";
      =     L 4.0;
      BLD   103;
      A     "Suska5_cor-";
      =     L 4.1;
      BLD   103;
      A     "Suska5_Pidtagnut";
      =     L 4.2;
      BLD   103;
      CALL  "Calc_Speed_Unit" , "CalcSpeed_Sushka5" (
           S_Privoda_pochatkova     := "Speed_KlajPress_R",
           Dodat_svidkist           := L 4.0,
           Vidnyat_svidkist         := L 4.1,
           Pidtyagnut               := L 4.2,
           Percent_In               := "Suchka5_Correction",
           S_Privoda_rozrah         := "Speed_Suchka5_R",
           Percent_Out              := "Suchka5_Correction");
      NOP   0;
NETWORK
TITLE = Розрахунок швидкості сушка 6
      A     "Suska6_cor+";
      =     L 4.0;
      BLD   103;
      A     "Suska6_cor-";
      =     L 4.1;
      BLD   103;
      A     "Suska6_Pidtagnut";
      =     L 4.2;
      BLD   103;
      CALL  "Calc_Speed_Unit" , "CalcSpeed_Sushka6" (
           S_Privoda_pochatkova     := "Speed_Suchka5_R",
           Dodat_svidkist           := L 4.0,
           Vidnyat_svidkist         := L 4.1,
           Pidtyagnut               := L 4.2,
           Percent_In               := "Suchka6_Correction",
           S_Privoda_rozrah         := "Speed_Suchka6_R",
           Percent_Out              := "Suchka6_Correction");
      NOP   0;
NETWORK
TITLE = Розрахунок швидкості сушка 7
      A(;
      A     "Suska7_cor+";
      =     L 4.0;
      BLD   103;
      A     "Suska7_cor-";
      =     L 4.1;
      BLD   103;
      A     "Suska7_Pidtagnut";
      =     L 4.2;
      BLD   103;
      CALL  "Calc_Speed_Unit" , "CalcSpeed_Sushka7" (
           S_Privoda_pochatkova     := "Speed_Suchka6_R",
           Dodat_svidkist           := L 4.0,
           Vidnyat_svidkist         := L 4.1,
           Pidtyagnut               := L 4.2,
           Percent_In               := "Suchka7_Correction",
           S_Privoda_rozrah         := "Speed_Suchka7_R",
           Percent_Out              := "Suchka7_Correction");
      A     BR;
      );
      JNB   _001;
      L     "Speed_Suchka7_R";
      T     "Signals_To_Nakat".Speed_Suchka7_di;
_001: NOP   0;
NETWORK
TITLE = Розрахунок швидкості каландр
      CALL  "Calc_Speed_Unit" , DB 141 (
           S_Privoda_pochatkova     := "Speed_Suchka7_R",
           S_Privoda_rozrah         := "Speed_Kalandr");
      NOP   0;
NETWORK
TITLE = Розрахунок швидкості накат
      CALL  "Calc_Speed_Unit" , DB 142 (
           S_Privoda_pochatkova     := "Speed_Kalandr",
           S_Privoda_rozrah         := "Speed_Nakat");
      NOP   0;
NETWORK
TITLE = Розрахунок швидкості паперо-ведучий вал 1
//*******************************************************
//
      A     "PaperVedVal1_Korec +";
      =     L 4.0;
      BLD   103;
      A     "PaperVedVal1_Korec -";
      =     L 4.1;
      BLD   103;
      CALL  "Calc_Speed_Unit" , "PapVed1_Speed_Unit" (
           S_Privoda_pochatkova     := "Speed_KombiPressR",
           Dodat_svidkist           := L 4.0,
           Vidnyat_svidkist         := L 4.1,
           Percent_In               := "PAPER_VED_1_KOEF_VIDHILU",
           S_Privoda_rozrah         := "Speed_PapVed1",
           Percent_Out              := "PAPER_VED_1_KOEF_VIDHILU");
      NOP   0;
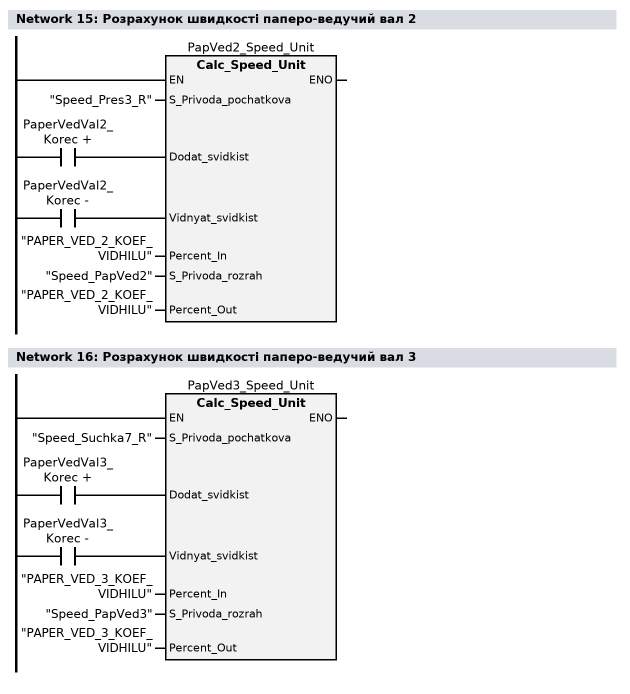
NETWORK
TITLE = Розрахунок швидкості паперо-ведучий вал 2
//*******************************************************
//
      A     "PaperVedVal2_Korec +";
      =     L 4.0;
      BLD   103;
      A     "PaperVedVal2_Korec -";
      =     L 4.1;
      BLD   103;
      CALL  "Calc_Speed_Unit" , "PapVed2_Speed_Unit" (
           S_Privoda_pochatkova     := "Speed_Pres3_R",
           Dodat_svidkist           := L 4.0,
           Vidnyat_svidkist         := L 4.1,
           Percent_In               := "PAPER_VED_2_KOEF_VIDHILU",
           S_Privoda_rozrah         := "Speed_PapVed2",
           Percent_Out              := "PAPER_VED_2_KOEF_VIDHILU");
      NOP   0;
NETWORK
TITLE = Розрахунок швидкості паперо-ведучий вал 3
//*******************************************************
//
      A     "PaperVedVal3_Korec +";
      =     L 4.0;
      BLD   103;
      A     "PaperVedVal3_Korec -";
      =     L 4.1;
      BLD   103;
      CALL  "Calc_Speed_Unit" , "PapVed3_Speed_Unit" (
           S_Privoda_pochatkova     := "Speed_Suchka7_R",
           Dodat_svidkist           := L 4.0,
           Vidnyat_svidkist         := L 4.1,
           Percent_In               := "PAPER_VED_3_KOEF_VIDHILU",
           S_Privoda_rozrah         := "Speed_PapVed3",
           Percent_Out              := "PAPER_VED_3_KOEF_VIDHILU");
      NOP   0;
END_FUNCTION

FUNCTION "RPM_Calculation" : VOID	// FC 11
VERSION : 0.1
BEGIN
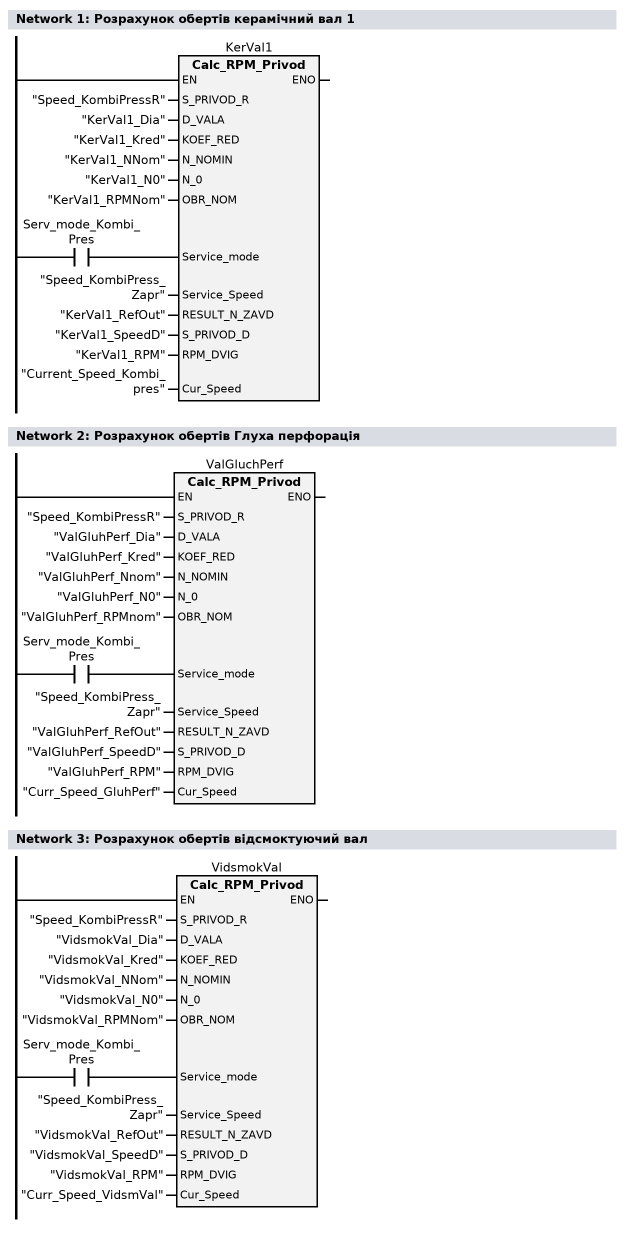
NETWORK
TITLE = Розрахунок обертів керамічний вал 1
      A     "Serv_mode_Kombi_Pres";
      =     L 0.0;
      BLD   103;
      CALL  "Calc_RPM_Privod" , "KerVal1" (
           S_PRIVOD_R               := "Speed_KombiPressR",
           D_VALA                   := "KerVal1_Dia",
           KOEF_RED                 := "KerVal1_Kred",
           N_NOMIN                  := "KerVal1_NNom",
           N_0                      := "KerVal1_N0",
           OBR_NOM                  := "KerVal1_RPMNom",
           Service_mode             := L 0.0,
           Service_Speed            := "Speed_KombiPress_Zapr",
           RESULT_N_ZAVD            := "KerVal1_RefOut",
           S_PRIVOD_D               := "KerVal1_SpeedD",
           RPM_DVIG                 := "KerVal1_RPM",
           Cur_Speed                := "Current_Speed_Kombi_pres");
      NOP   0;
NETWORK
TITLE = Розрахунок обертів Глуха перфорація
      A     "Serv_mode_Kombi_Pres";
      =     L 0.0;
      BLD   103;
      CALL  "Calc_RPM_Privod" , "ValGluchPerf" (
           S_PRIVOD_R               := "Speed_KombiPressR",
           D_VALA                   := "ValGluhPerf_Dia",
           KOEF_RED                 := "ValGluhPerf_Kred",
           N_NOMIN                  := "ValGluhPerf_Nnom",
           N_0                      := "ValGluhPerf_N0",
           OBR_NOM                  := "ValGluhPerf_RPMnom",
           Service_mode             := L 0.0,
           Service_Speed            := "Speed_KombiPress_Zapr",
           RESULT_N_ZAVD            := "ValGluhPerf_RefOut",
           S_PRIVOD_D               := "ValGluhPerf_SpeedD",
           RPM_DVIG                 := "ValGluhPerf_RPM",
           Cur_Speed                := "Curr_Speed_GluhPerf");
      NOP   0;
NETWORK
TITLE = Розрахунок обертів відсмоктуючий вал
      A     "Serv_mode_Kombi_Pres";
      =     L 0.0;
      BLD   103;
      CALL  "Calc_RPM_Privod" , "VidsmokVal" (
           S_PRIVOD_R               := "Speed_KombiPressR",
           D_VALA                   := "VidsmokVal_Dia",
           KOEF_RED                 := "VidsmokVal_Kred",
           N_NOMIN                  := "VidsmokVal_NNom",
           N_0                      := "VidsmokVal_N0",
           OBR_NOM                  := "VidsmokVal_RPMNom",
           Service_mode             := L 0.0,
           Service_Speed            := "Speed_KombiPress_Zapr",
           RESULT_N_ZAVD            := "VidsmokVal_RefOut",
           S_PRIVOD_D               := "VidsmokVal_SpeedD",
           RPM_DVIG                 := "VidsmokVal_RPM",
           Cur_Speed                := "Curr_Speed_VidsmVal");
      NOP   0;
